{attribute addProperty BoxType "EL3314-0002-0016"}
{attribute addProperty Id "StatusAT %I*Status_F0C7FE3C1621ValueAT %I*DINT32417"}
{attribute addProperty CRC "1552041520"}
{attribute addProperty SizeInBites "48"}
{attribute addProperty SizeInBytes "6"}
TYPE TC_Inputs_Channel_5C824630 :
STRUCT
	{attribute addProperty Name "Status"}
	Status AT %I* : Status_F0C7FE3C;
	{attribute addProperty Name "Value"}
	Value AT %I* : DINT;
END_STRUCT
END_TYPE

(* stored: Version 1.2.0.0, ProductVersion 3.1.4024.9
   DUT TC_Inputs_Channel_5C824630: Id {65770358-b3ad-4b04-9ad9-11a84602472a} *)
